// TwinCAT 3 PLC project DAD_Driver
// ProgramVersion: 3.1.4020.4
// libraries:
//   Tc2_Standard, * (Beckhoff Automation GmbH)
//   Tc2_System, * (Beckhoff Automation GmbH)
//   Tc3_Module, * (Beckhoff Automation GmbH)
// project tree:
//   990 - NTO Library/Barcode Readers/Base/ BarcodeCodeReadingResult.TcDUT, BarcodeReader.TcPOU, BarcodeReaderState.TcDUT, IBarcodeReader.TcIO, IBarcodeReaderSubscriber.TcIO
//   990 - NTO Library/Barcode Readers/Datalogic/ DAD_Controller.TcPOU, DatalogicOutputs.TcDUT, IDAD_Controller.TcIO, DAD_ControlFieldRecieve.TcDUT, DAD_ControlFieldTransmit.TcDUT, DatalogicInputs.TcDUT
//   990 - NTO Library/Data/ Data.TcDUT, IDataReciever.TcIO, IDataTransmit.TcIO
//   990 - NTO Library/HResult/ Busy.TcPOU, Fail.TcPOU, GetCode.TcPOU, HResultErrors.TcGVL, HResultSuccess.TcGVL, Success.TcPOU
//   990 - NTO Library/ NTO_LibraryAscii.TcGVL
//   990 - NTO Library/Object/ ErrorHistory.TcDUT, IObject.TcIO, Object.TcPOU, ObjectSetup.TcGVL
//   / MAIN.TcPOU, PlcTask.TcTTO
//   Test/ testData.TcDUT, TestRecieve.TcPOU
// real-time tasks:
//   TASK PlcTask: cycle T#5ms, priority 20, ADS port 350
// I/O:
//   DEVICE ProfinetController, AmsNetId 5.42.152.160.3.1
//     datalogic [HMS Industrial Networks This Device Access Point supports RT communication ABCC-PRT]
//       modules: Term 1 (DAP Module), Term 2 (Output 1 byte), Term 3 (Output 1 byte), Term 4 (Output 1 byte), Term 5 (Output 1 byte), Term 6 (Output 1 byte), Term 7 (Output 1 byte), Term 8 (Output 1 byte), Term 9 (Output 1 byte), Term 10 (Input 1 byte), Term 11 (Input 1 byte), Term 12 (Input 1 byte), Term 13 (Input 1 byte), Term 14 (Input 1 byte), Term 15 (Input 1 byte), Term 16 (Input 1 byte), Term 17 (Input 1 byte), Term 18 (Input 1 byte), Term 19 (Input 1 byte), Term 20 (Input 1 byte), Term 21 (Input 1 byte), Term 22 (Input 1 byte), Term 23 (Input 1 byte), Term 24 (Input 1 byte), Term 25 (Input 1 byte), Term 26 (Input 1 byte), Term 27 (Input 1 byte), Term 28 (Input 1 byte), Term 29 (Input 1 byte), Term 30 (Input 1 byte), Term 31 (Input 1 byte), Term 32 (Input 1 byte), Term 33 (Input 1 byte), Term 34 (Input 1 byte), Term 35 (Input 1 byte), Term 36 (Input 1 byte), Term 37 (Input 1 byte), Term 38 (Input 1 byte), Term 39 (Input 1 byte), Term 40 (Input 1 byte), Term 41 (Input 1 byte), Term 42 (Input 1 byte), Term 43 (Input 1 byte), Term 44 (Input 1 byte), Term 45 (Input 1 byte), Term 46 (Input 1 byte), Term 47 (Input 1 byte), Term 48 (Input 1 byte), Term 49 (Input 1 byte), Term 50 (Input 1 byte), Term 51 (Input 1 byte), Term 52 (Input 1 byte), Term 53 (Input 1 byte), Term 54 (Input 1 byte), Term 55 (Input 1 byte), Term 56 (Input 1 byte), Term 57 (Input 1 byte), Term 58 (Input 1 byte), Term 59 (Input 1 byte), Term 60 (Input 1 byte), Term 61 (Input 1 byte), Term 62 (Input 1 byte), Term 63 (Input 1 byte), Term 64 (Input 1 byte), Term 65 (Input 1 byte)
//   DEVICE Device 1 (EtherCAT)
// variable links:
//   DAD_Driver Instance <-> ProfinetController/datalogic
//     PlcTask Inputs/MAIN.inputMirror <-> API/Term 10 (Input 1 byte)/Subterm 1 (Input 1 byte)/Inputs/Input
//     PlcTask Inputs/MAIN.master.I_ApplicationDataRecieve[{0..51}] <-> API/Term {14..65} (Input 1 byte)/Subterm 1 (Input 1 byte)/Inputs/Input  (52 links)
//     PlcTask Inputs/MAIN.master.I_ControlFieldRecieve <-> API/Term 11 (Input 1 byte)/Subterm 1 (Input 1 byte)/Inputs/Input
//     PlcTask Inputs/MAIN.master.I_LengthFieldRecieve <-> API/Term 13 (Input 1 byte)/Subterm 1 (Input 1 byte)/Inputs/Input
//     PlcTask Inputs/MAIN.master.I_SAP_FieldRecieve <-> API/Term 12 (Input 1 byte)/Subterm 1 (Input 1 byte)/Inputs/Input
//     PlcTask Outputs/MAIN.master.Q_ApplicationDataTransmit[{0..3}] <-> API/Term {6..9} (Output 1 byte)/Subterm 1 (Output 1 byte)/Outputs/Output  (4 links)
//     PlcTask Outputs/MAIN.master.Q_ControlFieldTransmit <-> API/Term 3 (Output 1 byte)/Subterm 1 (Output 1 byte)/Outputs/Output
//     PlcTask Outputs/MAIN.master.Q_LengthFieldTransmit <-> API/Term 5 (Output 1 byte)/Subterm 1 (Output 1 byte)/Outputs/Output
//     PlcTask Outputs/MAIN.master.Q_SAP_FieldTransmit <-> API/Term 4 (Output 1 byte)/Subterm 1 (Output 1 byte)/Outputs/Output
//     PlcTask Outputs/MAIN.outputMirror <-> API/Term 2 (Output 1 byte)/Subterm 1 (Output 1 byte)/Outputs/Output

CONFIGURATION DAD_Driver
    RESOURCE PLC ON TwinCAT3
        TASK PlcTask(INTERVAL := T#5ms, PRIORITY := 20);
        PROGRAM MAIN WITH PlcTask : MAIN;
    END_RESOURCE
END_CONFIGURATION

// ---- 990 - NTO Library/Barcode Readers/Base/BarcodeCodeReadingResult.TcDUT
{attribute 'qualified_only'}
{attribute 'strict'}
///Reading result
TYPE BarcodeCodeReadingResult :
(
	noRead := 0,
    goodRead
);
END_TYPE

// ---- 990 - NTO Library/Barcode Readers/Base/BarcodeReaderState.TcDUT
{attribute 'qualified_only'}
{attribute 'strict'}
///Barcode reader state
TYPE BarcodeReaderState :
(
	unknown := 0, ///Unknown state
    resetting, //Resetting device
    noConnection, ///No connection to device
    standby, ///Standby and ready to activate
    reading, ///Reading
    gettingResult, ///Getting result from device
    evaluatingResult ///Evaluating the result from the device
);
END_TYPE

// ---- 990 - NTO Library/Barcode Readers/Datalogic/DatalogicOutputs.TcDUT
///Datalogic output control
TYPE DatalogicOutputs :
STRUCT
    output1 : BIT; //Output 1
    output2 : BIT; //Output 2
    output3 : BIT; //Output 3
    ourput4 : BIT; //Output 4
    reserved1 : BIT;
    reserved2 : BIT;
    reserved3 : BIT;
    phaseTrigger : BIT; //Reading phase trigger
END_STRUCT
END_TYPE

// ---- 990 - NTO Library/Barcode Readers/Datalogic/DAD_ControlFieldRecieve.TcDUT
///DAD Driver control field recieve
TYPE DAD_ControlFieldRecieve :
STRUCT
    TxBufferFull : BIT; //Toggles when Slave has made available new Input Area data
    RxBufferEmpty : BIT; //toggles when Output Area data has been read by Slave
    ResyncAcknowledge : BIT; //Set to 1 as an acknowledge to a resync request. With this bit, the master can detect a slave is on line.
    MoreBit : BIT; //is 1 when this is not the last piece of a fragmentation sequence while it is 0 when this is the last piece
    DAD_Fixed1 : BIT := FALSE; //Set to 0 when DAD messaging protocol is used
    DAD_Fixed2 : BIT := FALSE; //Set to 0 when DAD messaging protocol is used
    DAD_Fixed3 : BIT := FALSE; //Set to 0 when DAD messaging protocol is used
    DAD_Fixed4 : BIT := TRUE;  //Set to 1 when DAD messaging protocol is used  
END_STRUCT
END_TYPE

// ---- 990 - NTO Library/Barcode Readers/Datalogic/DAD_ControlFieldTransmit.TcDUT
///DAD Driver control field transmit
TYPE DAD_ControlFieldTransmit :
STRUCT
    TxBufferEmpty : BIT; //Must toggle when Input Area data has been read by Master
    RxBufferFull : BIT; //Must toggle when Master makes available new Output Area data
    ResyncRequest : BIT; //set to 1 for one second to resynchronize the slave. After resynchronization, all 4 handshake bits are set to 0
    MoreBit : BIT; //is 1 when this is not the last piece of a fragmentation sequence while it is 0 when this is the last piece
    DAD_Fixed1 : BIT := FALSE; //Set to 0 when DAD messaging protocol is used
    DAD_Fixed2 : BIT := FALSE; //Set to 0 when DAD messaging protocol is used
    DAD_Fixed3 : BIT := FALSE; //Set to 0 when DAD messaging protocol is used
    DAD_Fixed4 : BIT := TRUE;  //Set to 1 when DAD messaging protocol is used  
END_STRUCT
END_TYPE

// ---- 990 - NTO Library/Barcode Readers/Datalogic/DatalogicInputs.TcDUT
///Datalogic input mirroring
TYPE DatalogicInputs :
STRUCT
    input1 : BIT; //Mirror of input 1
    input2 : BIT; //Mirror of input 2
    input3 : BIT; //Mirror of input 3
    input4 : BIT; //Mirror of input 4
    reserved1 : BIT;
    reserved2 : BIT;
    reserved3 : BIT;
    phaseEcho : BIT; //Reading phase echo
END_STRUCT
END_TYPE

// ---- 990 - NTO Library/Data/Data.TcDUT
///Data result
TYPE Data :
STRUCT
    data : PVOID; ///Pointer to first byte of data
    length : UDINT; ///Data length
END_STRUCT
END_TYPE

// ---- 990 - NTO Library/Object/ErrorHistory.TcDUT
///Error history type
TYPE ErrorHistory : ARRAY[ObjectSetup.ErrorHistMin..ObjectSetup.ErrorHistMax] OF DWORD; END_TYPE

// ---- Test/testData.TcDUT
TYPE testData :
UNION
    buffer : ARRAY[0..9999] OF BYTE;
    bufferString : STRING[9998]; 
END_UNION
END_TYPE

// ---- 990 - NTO Library/HResult/HResultErrors.TcGVL
{attribute 'qualified_only'}
// HResult error types, in general HResult is error when less than 0
VAR_GLOBAL CONSTANT
    General : HRESULT := UDINT_TO_DINT(16#A0000000); //Fail with general error
    Busy : HRESULT :=  UDINT_TO_DINT(16#A0000001); //Function van't be called now, either other caller busy or other state is not allowing this function 
    InvalidParameter : HRESULT := UDINT_TO_DINT(16#A0000002); //Fail with invalid parameters    
	Connect : HRESULT := UDINT_TO_DINT(16#A0000003); //Fail, when trying to connect
	NotConnected : HRESULT := UDINT_TO_DINT(16#A0000004); //Fail, not connected
	AllocSocket : HRESULT := UDINT_TO_DINT(16#A0000005); //Fail, when allocating a socket
    InvalidPointerParameters : HRESULT := UDINT_TO_DINT(16#A0000006); //Fail, with invalid pointer parameters
END_VAR

// ---- 990 - NTO Library/HResult/HResultSuccess.TcGVL
{attribute 'qualified_only'}
// HResult success types, in general HResult is success when greather than equal 0
VAR_GLOBAL CONSTANT
    Done : HRESULT := 16#20000001; //Successfully done
    Busy : HRESULT := 16#20000002; //Busy, keep calling to wait for done or error    
END_VAR

// ---- 990 - NTO Library/NTO_LibraryAscii.TcGVL
{attribute 'qualified_only'}
//General control ascii charachters
VAR_GLOBAL CONSTANT
    STX	  : BYTE := 16#02; //Start of text
    ETX   : BYTE := 16#03; //End of text
    Space : BYTE := 16#20; //Space
	CR	  : BYTE := 16#0D; //Carriage return
	LF	  : BYTE := 16#0A; //Line feed
END_VAR

// ---- 990 - NTO Library/Object/ObjectSetup.TcGVL
{attribute 'qualified_only'}
VAR_GLOBAL CONSTANT
    ErrorHistMin : INT := 0; ///Error history array bound minimum
    ErrorHistMax : INT := 10; ///Error history array bound maximum
END_VAR

// ---- 990 - NTO Library/Barcode Readers/Base/IBarcodeReader.TcIO
///Interface for barcode readers
INTERFACE IBarcodeReader EXTENDS IObject

///End the reading
METHOD EndReading : HRESULT
VAR_OUTPUT
END_VAR
END_METHOD

/// Gets the state of optional digital inputs
PROPERTY GetDigitalInputs : ARRAY[0..7] OF BOOL
GET
END_GET
END_PROPERTY


PROPERTY GetState : BOOL
GET
END_GET
SET
END_SET
END_PROPERTY

///Get the last reading result
PROPERTY LastResult : Data
GET
END_GET
END_PROPERTY

///Reset the device
METHOD ResetDevice : HRESULT
VAR_INPUT
END_VAR
END_METHOD

/// Sets the state of digital outputs
METHOD SetDigitalOutputs : HRESULT
VAR_INPUT
    no : USINT; ///Output number to set between 0 - 7
    value : BOOL; ///Value to set output number
END_VAR
END_METHOD

///Start the reading
METHOD StartReading : HRESULT
VAR_INPUT
END_VAR
END_METHOD

///Get or set the subscriber to the barcode reader
PROPERTY Subscriber : IBarcodeReaderSubscriber
GET
END_GET
SET
END_SET
END_PROPERTY

END_INTERFACE

// ---- 990 - NTO Library/Barcode Readers/Base/IBarcodeReaderSubscriber.TcIO
///Interface for barcode readers result subscriber
INTERFACE IBarcodeReaderSubscriber

// New data recieved
METHOD NewDataRecieved : HResult
VAR_INPUT
    data : Data; ///Data recieved
    result : BarcodeCodeReadingResult; ///Reading result
END_VAR
END_METHOD

END_INTERFACE

// ---- 990 - NTO Library/Barcode Readers/Datalogic/IDAD_Controller.TcIO
INTERFACE IDAD_Controller EXTENDS IObject, IDataTransmit

///Flushes the data in the slave queue, must be called until HResult is not busy 
METHOD FlushData : HResult
VAR_IN_OUT
    id : UDINT; ///Used to id the called, should be 0 at first call, when functions finish normally success or error it will reset to 0
END_VAR
END_METHOD

//Resync the DAD controller driver
METHOD Resync : HResult
VAR_IN_OUT
    id : UDINT; ///Used to id the called, should be 0 at first call, when functions finish normally success or error it will reset to 0
END_VAR
END_METHOD

END_INTERFACE

// ---- 990 - NTO Library/Data/IDataReciever.TcIO
///Data reciever interface, implement this interface in the block
///that has to recieve data 
INTERFACE IDataReciever

// New data recieved
METHOD NewDataRecieved : HResult
VAR_INPUT
    data : Data; ///Data recieved
END_VAR
END_METHOD

END_INTERFACE

// ---- 990 - NTO Library/Data/IDataTransmit.TcIO
///Data trasnmitter interface, implemented by classes that can transmit data 
INTERFACE IDataTransmit EXTENDS IObject

// Gets the maximum allow data to send in one transmittion
PROPERTY MaxDataLength : UDINT
GET
END_GET
END_PROPERTY

/// Transmit data, keep calling while HResult returns busy
/// General implementation should fully copy data to internal
/// buffer at first call
METHOD TransmitData : HResult
VAR_INPUT
    data : Data; //Data to transmit
END_VAR
VAR_IN_OUT
    id : UDINT; ///Used to id the called, should be 0 at first call, when functions finish normally success or error it will reset to 0
END_VAR
END_METHOD

END_INTERFACE

// ---- 990 - NTO Library/Object/IObject.TcIO
///Base object interface
INTERFACE IObject

///Name
PROPERTY FINAL ClassName : STRING(50)
GET
END_GET
END_PROPERTY

//Cycle Task, do not override this methode cyclic code is placed in M_Control
METHOD CycleTask
VAR_INPUT
END_VAR
END_METHOD

///Error, do not implement property override
PROPERTY Error : BOOL
GET
END_GET
END_PROPERTY

///Error id, do not implement property override
PROPERTY ErrorID : DWORD
GET
END_GET
END_PROPERTY

(*Pointer to error history, do not implement property override*)
PROPERTY Errors : POINTER TO ErrorHistory
GET
END_GET
END_PROPERTY

///Reset error, allways call super
METHOD Reset
VAR_INPUT
END_VAR
END_METHOD

///Version,do not implement property override
PROPERTY PUBLIC Version : String(8)
GET
END_GET
END_PROPERTY

END_INTERFACE

// ---- MAIN.TcPOU
PROGRAM MAIN
VAR
    masterRecieve : TestRecieve;
    master : DAD_Controller(callback := masterRecieve, maxApplicationInputSize := 52, maxApplicationOutputSize := 4);
    sendMaster : ARRAY[0..255] OF BYTE;
    lengthMaster : UDINT;
    sendToMaster : BOOL;
    idMaster : UDINT;
    resetTestBuffer : BOOL;
END_VAR
VAR
    inputMirror AT %I* : BYTE;
    outputMirror AT %Q* : BYTE;
    trigScanner : BOOL;
END_VAR
VAR
    barcodeReader : BarcodeReader;
END_VAR

IF lengthMaster > 0 AND sendToMaster THEN
    IF master.TransmitData(data := ADR(sendMaster[0]), length := lengthMaster,id := idMaster) <> HResultSuccess.Busy THEN
        sendToMaster := FALSE;
	END_IF
END_IF

master.CycleTask();
outputMirror.7 := trigScanner;

IF resetTestBuffer THEN
    masterRecieve.Reset();
    resetTestBuffer := FALSE;
END_IF

END_PROGRAM

// ---- Test/TestRecieve.TcPOU
FUNCTION_BLOCK TestRecieve EXTENDS Object IMPLEMENTS IDataReciever
VAR
    buffer : testData;
    currentLength : UDINT;
END_VAR

{attribute '''NORMAL__COMMENT' := ' New data recieved'}
(* New data recieved*)
METHOD NewDataRecieved : HResult
VAR_INPUT
	data	: Data; //Data recieved
END_VAR
IF currentLength + data.length > 9999 THEN
    currentLength := 0;
END_IF

Tc2_System.MEMCPY(destAddr := ADR(buffer.buffer[currentLength]),srcAddr := data.data, n := data.length); 

currentLength := currentLength + data.length;
END_METHOD

(*Reset error, allways call super*)
METHOD Reset
Tc2_System.MEMSET(destAddr := ADR(buffer), fillByte := 0, n := SIZEOF(buffer));
currentLength := 0;
END_METHOD

END_FUNCTION_BLOCK

// ---- 990 - NTO Library/Object/Object.TcPOU
///Object base class for all classes
FUNCTION_BLOCK Object IMPLEMENTS IObject
VAR
    _className : STRING(50) := 'Object'; //Class name
    _version : STRING(8) := '1.0'; //Version
    firstPass : BOOL := FALSE; //First pass done
    _error : BOOL := FALSE; //Error
    _errorID : DWORD := 0; //Error id
    _errors : ErrorHistory; //Error history
END_VAR

///Add error to error history
METHOD PROTECTED AddError
VAR_INPUT
	errorID : DWORD; //Error ID
END_VAR
VAR
	addErrorLoop : INT;
END_VAR
FOR addErrorLoop := ObjectSetup.ErrorHistMax TO (ObjectSetup.ErrorHistMin + 1) BY -1 DO
	_errors[addErrorLoop] := _errors[addErrorLoop - 1];
END_FOR
_errors[ObjectSetup.ErrorHistMin] := errorID;
END_METHOD

(*Name, do not implement property override*)
PROPERTY ClassName : STRING(50)
GET
ClassName := _className;
END_GET
END_PROPERTY

///Control, override to get cyclic task in FB
METHOD INTERNAL Control
VAR_INPUT
END_VAR
END_METHOD

//Cycle Task, do not override this methode cyclic code is placed in M_Control 
METHOD FINAL CycleTask
IF NOT(firstPass) THEN
    firstPass := Init() = HResultSuccess.Done;
    IF NOT(firstPass) THEN
        RETURN;
	END_IF
END_IF
Control();
END_METHOD

(*Error, do not implement property override*)
PROPERTY Error : BOOL
GET
Error := _error;
END_GET
END_PROPERTY

(*error id, do not implement property override*)
PROPERTY ErrorID : DWORD
GET
ErrorID := _errorID;
END_GET
END_PROPERTY

(*Pointer to error history, do not implement property override*)
PROPERTY Errors : POINTER TO ErrorHistory
GET
Errors := ADR(_errors);
END_GET
END_PROPERTY

METHOD FB_init : BOOL
VAR_INPUT
	bInitRetains : BOOL; // if TRUE, the retain variables are initialized (warm start / cold start)
	bInCopyCode : BOOL;  // if TRUE, the instance afterwards gets moved into the copy code (online change)
END_VAR
firstPass := FALSE;
END_METHOD

///Initialize FB, Override to do custom initialize, no need to call super
METHOD INTERNAL Init : HRESULT
Init := HResultSuccess.Done;
END_METHOD

(*Reset error, allways call super*)
METHOD Reset
_error := FALSE;
_errorID := 0;
END_METHOD

///Set error on the Object and add entry to error history
METHOD PROTECTED SetError
VAR_INPUT
	errorID : DWORD; //Error ID
END_VAR
VAR
    setErrorLoop : INT;
END_VAR
IF NOT(_error) THEN
	_error := TRUE;
	THIS^._errorID := errorID;
	FOR setErrorLoop := ObjectSetup.ErrorHistMax TO (ObjectSetup.ErrorHistMin + 1) BY -1 DO
    	_errors[setErrorLoop] := _errors[setErrorLoop - 1];
	END_FOR
	_errors[ObjectSetup.ErrorHistMin] := _errorID;
END_IF
END_METHOD

(*Version,do not implement property override*)
PROPERTY Version : STRING(8)
GET
Version := _version;
END_GET
END_PROPERTY

END_FUNCTION_BLOCK

// ---- 990 - NTO Library/Barcode Readers/Datalogic/DAD_Controller.TcPOU
/// Controls a device using the Datalogic DAD driver.
/// The data is transferred using the Datalogic FCM DAD driver and 
/// gives the functions for resync and flush data.
/// A internal buffer of 256 butes allows for sending telegrams up
/// to that size in one transmittion. Telegram is automatically fragmnented
/// using Datalogic DAD driver standard.
FUNCTION_BLOCK DAD_Controller EXTENDS Object IMPLEMENTS IDAD_Controller
//---------------- DAD device connection ---------------------
VAR
    //---------------- Inputs from DAD device ----------------
    I_ControlFieldRecieve AT %I* : DAD_ControlFieldRecieve; ///Control field recieve
    I_SAP_FieldRecieve AT %I* : BYTE; //Service Access Protocol field recieve
    I_LengthFieldRecieve AT %I* : BYTE; //Data length recieve 
    I_ApplicationDataRecieve AT %I* : ARRAY[0..255] OF BYTE; //Application data recieve
    //---------------- Outputs to DAD device ----------------
    Q_ControlFieldTransmit AT %Q* : DAD_ControlFieldTransmit; ///Control field transmit
    Q_SAP_FieldTransmit AT %Q* : BYTE; //Service Access Protocol field transmit
    Q_LengthFieldTransmit AT %Q* : BYTE; //Data length transmit 
    Q_ApplicationDataTransmit AT %Q* : ARRAY[0..255] OF BYTE; //Application data recieve
END_VAR
//---------------- Class setup ---------------------
VAR
    _callback : IDataReciever; //Data reciever callback handler
    _maxApplicationInputSize : INT := 53; //Maximum application input size
    _maxApplicationOutputSize : INT := 5; //Maximum application output size
END_VAR
//---------------- Reciever ---------------------
VAR
    recieveBuffer : ARRAY[0..recieveMaxBufferLength] OF BYTE; //Recieve buffer
    recieveBufferLength : UDINT; //Current buffer length
    recieveWatchdog : Tc2_Standard.TON; //Timeout for recieving active
    _recieveTimeout : TIME := T#10S; //Watchdog time
END_VAR
VAR CONSTANT
    recieveMaxBufferLength : UDINT := 255; // Recieve buffer max length
END_VAR
//---------------- Transmitter ---------------------
VAR
    transmitBuffer : ARRAY[0..transmitMaxBufferLength] OF BYTE; //Send buffer
    transmitBufferLength : UDINT; //Current buffer length
    transmittedLength : UDINT; //Fragments length transmitted
    currentTransmitCallState : UDINT := 0; // Current transmit call state
    transmitting : BOOL; //Currently transmitting
    transmitWatchdog : Tc2_Standard.TON; //Timeout for recieving active
    _transmitTimeout : TIME := T#10S; //Watchdog time
END_VAR
VAR CONSTANT
    transmitMaxBufferLength : UDINT := 50; // Transmit buffer max length
END_VAR
//---------------- Resync ---------------------
VAR
    currentResyncCallState : UDINT := 0; // Current resync call state
    resyncWatchdog : Tc2_Standard.TON; //Watchdog
    resyncTimeout : TIME := T#10S; //Watchdog time
END_VAR
//---------------- Flush ----------------------
VAR
    currentFlushCallState : UDINT := 0; // Current flush call state
    flushWatchdog : Tc2_Standard.TON; //Watchdog
    flushTimeout : TIME := T#10S; //Watchdog time
END_VAR

///Control, override to get cyclic task in FB
METHOD INTERNAL Control
IF currentResyncCallState = 0 THEN
    Reciever();
END_IF
Transmitter();

// --------------- Resync watchdog ---------------
resyncWatchdog(IN := currentResyncCallState <> 0, PT := resyncTimeout);
IF resyncWatchdog.Q THEN
    currentResyncCallState := 0;
    Q_ControlFieldTransmit.ResyncRequest := FALSE;
END_IF
// -------------- Flush watchdog -----------------
flushWatchdog(IN := currentFlushCallState <> 0, PT := flushTimeout);
IF flushWatchdog.Q THEN
    currentFlushCallState := 0;
END_IF
END_METHOD

METHOD FB_init : BOOL
VAR_INPUT
	bInitRetains : BOOL; // if TRUE, the retain variables are initialized (warm start / cold start)
	bInCopyCode : BOOL;  // if TRUE, the instance afterwards gets moved into the copy code (online change)
    callback : IDataReciever; //Calling function block
    maxApplicationInputSize : INT := 53; //Maximum application input size
    maxApplicationOutputSize : INT := 5; //Maximum application output size
END_VAR
THIS^._version := '1.0';
THIS^._className := 'DAD_Controller';
THIS^._callback := callback;
THIS^._maxApplicationInputSize := maxApplicationInputSize;
THIS^._maxApplicationOutputSize := maxApplicationOutputSize;
END_METHOD

///Flushes the data in the slave queue, must be called until HResult is not busy 
METHOD FlushData : HResult
VAR_IN_OUT
    id : UDINT; ///Used to id the called, should be 0 at first call, when functions finish normally success or error it will reset to 0
END_VAR
VAR CONSTANT
    flushID : UDINT := 10003; //Unique function call id
END_VAR
END_METHOD

// Gets the maximum allow data to send in one transmittion
PROPERTY MaxDataLength : UDINT
GET
MaxDataLength := transmitMaxBufferLength;
END_GET
END_PROPERTY

METHOD PROTECTED Reciever
VAR
    data : Data;
END_VAR
//---------------- Recieve new data from slave ---------------------
IF I_ControlFieldRecieve.TxBufferFull <> Q_ControlFieldTransmit.TxBufferEmpty THEN
    IF (I_LengthFieldRecieve + recieveBufferLength) >= recieveMaxBufferLength THEN
        THIS^.SetError(errorID := 1);
    ELSE
        Tc2_System.MEMCPY(destAddr := ADR(recieveBuffer[recieveBufferLength]), srcAddr := ADR(I_ApplicationDataRecieve[0]), n := BYTE_TO_UDINT(I_LengthFieldRecieve));
        recieveBufferLength := recieveBufferLength + I_LengthFieldRecieve;
        IF recieveBufferLength >= recieveMaxBufferLength THEN
            recieveBufferLength := recieveMaxBufferLength;
        END_IF
	END_IF
    // Check if further message fragments, if full message send to callback else add to buffer and wait
    // for next message fragment 
    IF NOT(I_ControlFieldRecieve.MoreBit) THEN
        IF _callback <> 0 THEN
            data.data := ADR(recieveBuffer[0]);
            data.length := recieveBufferLength;
            _callback.NewDataRecieved(data := data);
		END_IF
        recieveBufferLength := 0;
    END_IF
    Q_ControlFieldTransmit.TxBufferEmpty := I_ControlFieldRecieve.TxBufferFull;
END_IF
//--------------------- Watchdog ---------------------------
recieveWatchdog(IN := recieveBufferLength > 0, PT := _recieveTimeout);
IF recieveWatchdog.Q THEN
    recieveBufferLength := 0;
    THIS^.AddError(errorID := 2);
END_IF
END_METHOD

PROPERTY RecieveTimeout : TIME
GET
RecieveTimeout := _recieveTimeout;
END_GET
SET
_recieveTimeout := RecieveTimeout;
END_SET
END_PROPERTY

//Resync the DAD controller driver
METHOD Resync : HResult
VAR_IN_OUT
    id : UDINT; ///Used to id the called, should be 0 at first call, when functions finish normally success or error it will reset to 0
END_VAR
VAR CONSTANT
    resyncID : UDINT := 10002; //Unique function call id
END_VAR
// ---------------- Check function call ---------------------
IF currentResyncCallState <> 0 AND id = 0 THEN
    Resync := HResultErrors.Busy;
    RETURN;
END_IF
IF currentResyncCallState = 0 AND id <> 0 THEN
    Resync := HResultErrors.InvalidParameter;
    RETURN;
END_IF
IF id <> 0 AND id <> resyncID THEN
    Resync := HResultErrors.InvalidParameter;
    RETURN;
END_IF
Resync := HResultSuccess.Busy;
//Start the resync process at first call
IF currentResyncCallState = 0 AND id = 0 THEN    
    currentResyncCallState := resyncID;
    id := currentResyncCallState;
    Q_ControlFieldTransmit.ResyncRequest := TRUE;
END_IF
IF Q_ControlFieldTransmit.ResyncRequest AND I_ControlFieldRecieve.ResyncAcknowledge THEN
    Q_ControlFieldTransmit.ResyncRequest := FALSE;
END_IF
IF NOT Q_ControlFieldTransmit.ResyncRequest AND NOT I_ControlFieldRecieve.ResyncAcknowledge THEN
    Q_ControlFieldTransmit.MoreBit := FALSE;
    Q_ControlFieldTransmit.RxBufferFull := FALSE;
    Q_ControlFieldTransmit.TxBufferEmpty := FALSE;
    recieveBufferLength := 0;
    currentTransmitCallState := 0;
    transmitBufferLength := 0;
    transmitting := FALSE;
    THIS^.Reset();
    id := 0;
    currentResyncCallState := 0;
    Resync := HResultSuccess.Done;
END_IF;
END_METHOD

/// Transmit data, keep calling while HResult returns busy
/// General implementation should fully copy data to internal
/// buffer at first call
METHOD TransmitData : HResult
VAR_INPUT
    data : PVOID; ///Pointer to first byte of data to send
    length : UDINT; ///Data length to send
END_VAR
VAR_IN_OUT
    id : UDINT; ///Used to id the called, should be 0 at first call, when functions finish normally success or error it will reset to 0
END_VAR
VAR CONSTANT
    transmitID : UDINT := 10001; //Unique function call id
END_VAR
// ---------------- Check function call ---------------------
IF currentTransmitCallState <> 0 AND id = 0 THEN
    TransmitData := HResultErrors.Busy;
    RETURN;
END_IF
IF currentTransmitCallState = 0 AND id <> 0 THEN
    TransmitData := HResultErrors.InvalidParameter;
    RETURN;
END_IF
IF id <> 0 AND id <> transmitID THEN
    TransmitData := HResultErrors.InvalidParameter;
    RETURN;
END_IF
IF currentResyncCallState <> 0 THEN
   TransmitData := HResultErrors.NotConnected;
   RETURN; 
END_IF

// At first call, copy new telegram to buffer
IF id = 0 AND currentTransmitCallState = 0 THEN
    IF data = 0 OR length = 0 OR length >= transmitMaxBufferLength THEN
        TransmitData := HResultErrors.InvalidPointerParameters;
        RETURN;
    END_IF
    id := transmitID;
    currentTransmitCallState := transmitID;
    TransmitData := HResultSuccess.Busy;
    Tc2_System.MEMCPY(destAddr := ADR(transmitBuffer), srcAddr := data, n := length);
    transmitBufferLength := length;
    transmitting := FALSE;
END_IF
// Transmit data string
IF id = currentTransmitCallState THEN
    TransmitData := HResultSuccess.Busy;
    IF NOT(transmitting) THEN
        IF I_ControlFieldRecieve.RxBufferEmpty = Q_ControlFieldTransmit.RxBufferFull THEN
            /// Transmit data fragment
            transmitting := TRUE;
            Q_LengthFieldTransmit := UDINT_TO_BYTE(MIN(INT_TO_UDINT(_maxApplicationOutputSize), transmitBufferLength - transmittedLength));
            Q_ControlFieldTransmit.MoreBit := (transmittedLength + Q_LengthFieldTransmit) < transmitBufferLength;
            Tc2_System.MEMCPY(destAddr := ADR(Q_ApplicationDataTransmit), srcAddr := ADR(transmitBuffer[transmittedLength]), n := Q_LengthFieldTransmit);
            transmittedLength := transmittedLength + Q_LengthFieldTransmit;
            Q_ControlFieldTransmit.RxBufferFull := NOT Q_ControlFieldTransmit.RxBufferFull;
		END_IF
    ELSE    
       IF I_ControlFieldRecieve.RxBufferEmpty = Q_ControlFieldTransmit.RxBufferFull THEN
           IF transmittedLength >= transmitBufferLength THEN
               TransmitData := HResultSuccess.Done;
               transmittedLength := 0;
               currentTransmitCallState := 0;
               id := 0;
		   END_IF
           transmitting := FALSE;
	   END_IF
	END_IF
END_IF
END_METHOD

METHOD PROTECTED Transmitter
//--------------------- Watchdog ---------------------------
transmitWatchdog(IN := currentTransmitCallState <> 0, PT := _transmitTimeout);
IF transmitWatchdog.Q THEN
    currentTransmitCallState := 0;
    transmitBufferLength := 0;
    transmitting := 0;
    THIS^.AddError(errorID := 3);
END_IF
END_METHOD

PROPERTY TransmitTimeout : TIME
GET
TransmitTimeout := _transmitTimeout;
END_GET
SET
_transmitTimeout := TransmitTimeout;
END_SET
END_PROPERTY

END_FUNCTION_BLOCK

// ---- 990 - NTO Library/HResult/Busy.TcPOU
///Checks if the returned HRESULT is success and busy
FUNCTION Busy : BOOL
VAR_INPUT
    hr : HRESULT;
END_VAR
VAR
END_VAR

Busy := (hr = HResultSuccess.Busy);

END_FUNCTION

// ---- 990 - NTO Library/Barcode Readers/Base/BarcodeReader.TcPOU
FUNCTION_BLOCK BarcodeReader EXTENDS Object IMPLEMENTS IBarcodeReader, IDataReciever
VAR
END_VAR

///Control, override to get cyclic task in FB
METHOD INTERNAL Control
END_METHOD

///End the reading
METHOD EndReading : HRESULT
VAR_OUTPUT
END_VAR
END_METHOD

METHOD FB_init : BOOL
VAR_INPUT
	bInitRetains : BOOL; // if TRUE, the retain variables are initialized (warm start / cold start)
	bInCopyCode : BOOL;  // if TRUE, the instance afterwards gets moved into the copy code (online change)
END_VAR
_version := '1.0';
_className := 'BarcodeReader';
END_METHOD

/// Gets the state of optional digital inputs
PROPERTY GetDigitalInputs : ARRAY[0..7] OF BOOL
GET
END_GET
END_PROPERTY


PROPERTY GetState : BOOL
GET
END_GET
SET
END_SET
END_PROPERTY

///Get the last reading result
PROPERTY LastResult : Data
GET
END_GET
END_PROPERTY

// New data recieved
METHOD NewDataRecieved : HResult
VAR_INPUT
    data : Data; ///Data recieved
END_VAR
END_METHOD

///Reset the device
METHOD ResetDevice : HRESULT
VAR_INPUT
END_VAR
END_METHOD

/// Sets the state of digital outputs
METHOD SetDigitalOutputs : HRESULT
VAR_INPUT
    no : USINT; ///Output number to set between 0 - 7
    value : BOOL; ///Value to set output number
END_VAR
END_METHOD

///Start the reading
METHOD StartReading : HRESULT
VAR_INPUT
END_VAR
END_METHOD

///Get or set the subscriber to the barcode reader
PROPERTY Subscriber : IBarcodeReaderSubscriber
GET
END_GET
SET
END_SET
END_PROPERTY

END_FUNCTION_BLOCK

// ---- 990 - NTO Library/HResult/Fail.TcPOU
///Checks if the HRESULT is error
FUNCTION Fail : BOOL
VAR_INPUT
    hr : HRESULT;
END_VAR
VAR
END_VAR

Fail := (hr < 0);

END_FUNCTION

// ---- 990 - NTO Library/HResult/Success.TcPOU
///Checks if the returned HRESULT is success
FUNCTION Success : BOOL
VAR_INPUT
    hr : HRESULT;
END_VAR
VAR
END_VAR

Success := (hr >= 0);

END_FUNCTION

// ---- 990 - NTO Library/HResult/GetCode.TcPOU
///Get the Code from the HRESULT
FUNCTION GetCode : UINT
VAR_INPUT
    hr : HRESULT;
END_VAR
VAR
END_VAR

GetCode := UDINT_TO_UINT(DINT_TO_UDINT(hr) AND 16#0000FFFF);

END_FUNCTION
